# EPICS StreamDevice protocol: iocs/rpi-beamtable/beamtable_serial.proto
Terminator = CR LF;

ReadTimeout = 1000;
#WriteTimeout = 100;
#PollPeriod = 400;

ExtraInput = Ignore;

# serial device returns the adc values as long data type. Also the values are in micro volts

setPos {
	out "%f";
}

getPos {
	in "adcpos%f";
}

motor_status {
	in "0s%i";
}

motor_direction {
	in "1s%i";
}
